Staubli VAL3: checkColValue.pgx

public program checkColValue(string x_sColCharac (dimensions=1), bool& x_bColOk[] (dimensions=1))
begin
  //-----------------------------------------------------------------------
  //Header begin
  //Description of program
  //  Check the column number of the x_sCellNumber.
  //
  // Input Parameters
  //   x_sCellNumber  :
  //     role : cell number in string format.
  //            Must be : - First digit is a letter (A-Z) for Column number
  //                      - 3 next digits is a number for Row number
  //
  // Output Parameteres
  //  x_bColOk  :
  //    role : returns true if the operation succeeded and false
  //          otherwise
  //
  //Header end
  //-----------------------------------------------------------------------

  //Verify column character (between "A" to "Z" or "a" to "z")
  x_bColOk=(asc(x_sColCharac,0)>=asc("a",0)) and (asc(x_sColCharac,0)<=asc("z",0))
  x_bColOk=x_bColOk or (asc(x_sColCharac,0)>=asc("A",0)) and (asc(x_sColCharac,0)<=asc("Z",0))
end
